Omron Sysmac Studio project ToggleButton (Sysmac Studio 1.65.0.64007, StandardProject)

# Controller new_Controller_0: NX1P2-1040DT1 version 1.69
Task PrimaryTask (priority 4, period or condition 2000): Program0



PROGRAM Program0
VAR
    ToggleButton : BOOL;
    T1 : BOOL;
    T2 : BOOL;
    T3 : BOOL;
    T4 : BOOL;
    MotorCikis : BOOL;
    MotorStart : BOOL;
END_VAR

(* Section Section0: ladder, written here as Structured Text *)

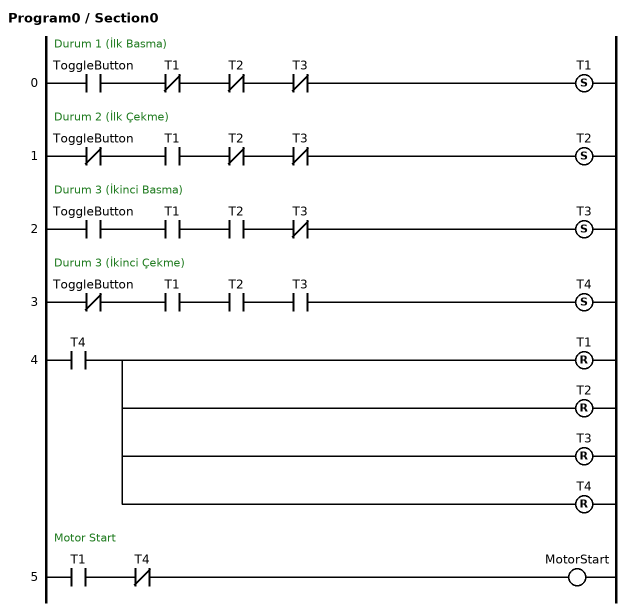
(* Rung 0: Durum 1 (İlk Basma) *)
IF ToggleButton AND NOT T1 AND NOT T2 AND NOT T3 THEN T1 := TRUE; END_IF;
(* Rung 1: Durum 2 (İlk Çekme) *)
IF NOT ToggleButton AND T1 AND NOT T2 AND NOT T3 THEN T2 := TRUE; END_IF;
(* Rung 2: Durum 3 (İkinci Basma) *)
IF ToggleButton AND T1 AND T2 AND NOT T3 THEN T3 := TRUE; END_IF;
(* Rung 3: Durum 3 (İkinci Çekme) *)
IF NOT ToggleButton AND T1 AND T2 AND T3 THEN T4 := TRUE; END_IF;
(* Rung 4 *)
IF T4 THEN
    T1 := FALSE;
    T2 := FALSE;
    T3 := FALSE;
    T4 := FALSE;
END_IF;
(* Rung 5: Motor Start *)
MotorStart := T1 AND NOT T4;
END_PROGRAM